PROGRAM MAIN
VAR
	bInit:					BOOL:=TRUE;	
END_VAR

INIT_DataSet();
RECIPE_Controller();
DRIVE_Controller();

(*
	Fill the recipie variables 
		#CMD is represent IsCOMMAND
		XXX 3 digit integer represent the JigID
		XXX 3 digit integer represent the Command type
		
		Example:
		#CMD000000#END									- START OF SEQUENCE (No PARAMETER)
		#CMD999999#END									- END OF SEQUENCE (No PARAMETER)
		#CMD001000#END 									- EXECUTE THE No.:0 ADAPTER SEQUENCE (No PARAMETER)
		#CMD001005#END 									- EXECUTE THE No.:5 ADAPTER SEQUENCE (No PARAMETER)
		#CMD001015#PARAM:125.1265#END					- EXECUTE THE No.:5 ADAPTER SEQUENCE (With PARAMETER)
		#CMD001100#POS:1#END							- GO TO POSITION
		#CMD001110#POS:1#SCREW:2#SCREWPRG:26#END		- GO TO POSITION
*)
IF bInit THEN
	RECIPE.SequenceArray:= __NEW(STRING, 10);	
	RECIPE.SequenceArray[0]:='#CMD000000#END'; 			
	RECIPE.SequenceArray[1]:='#CMD001100#POS:0#END';
	RECIPE.SequenceArray[2]:='#CMD001100#POS:1#END';
	RECIPE.SequenceArray[3]:='#CMD001005#POS:2#END';
	RECIPE.SequenceArray[4]:='#CMD001100#POS:3#END';
	RECIPE.SequenceArray[5]:='#CMD001100#POS:4#END';
	RECIPE.SequenceArray[6]:='#CMD001003#POS:5#END';
	RECIPE.SequenceArray[7]:='#CMD001100#POS:6#END';
	RECIPE.SequenceArray[8]:='#CMD001100#POS:7#END';
	RECIPE.SequenceArray[9]:='#CMD999999#END';	
	bInit:=FALSE;		
END_IF

END_PROGRAM

(* stored: Version 1.1.0.1, ProductVersion 3.1.4022.18
   POU MAIN: Id {015a52a7-5bf1-4c05-ba26-f68ec63d8824}, SpecialFunc None *)
